PROGRAM Read_TrailerID
VAR
	Trailer_ID AT %I*	: UINT;
END_VAR

;

END_PROGRAM

(* stored: Version 1.1.0.1, ProductVersion 3.1.4024.6
   POU Read_TrailerID: Id {e1372c7c-abe8-4077-94d5-6aa297d659bb}, SpecialFunc None *)
